# EPICS autosave request: ADApp/Db/NDRateLimit_settings.req
$(P)$(R)Mode
$(P)$(R)Limit
file "NDPluginBase_settings.req", P=$(P), R=$(R)
